PROGRAM prgVar
VAR
	fbVar			: FB_VarInfo_V3;
	fbrw1			: FB_ReadWrite_V2;
END_VAR

fbVar(
	bReadInfo:= , 
	eTMCFile:= eSelectTMCFile.eDontUseTMCFile, 
	eSavePositionTMCFile:= eSavePositionOnPLC.ePostionC, 
	udiCounterFoundVariables=> , 
	bError=> , 
	bBusy=> , 
	byProgress=> , 
	udiErrorCodeOut=> , 
	eErrorVarInfo_Out=> , 
	sVarWithError=> );
fbVar();
fbVar();	

fbRW1(	eUploadType := eSelectDataUploadType.e_Change_Intervall5min,
		bBusy=> , 
		bError=> , 
		udiErrorCodeOut=> , 
		eErrorReadWrite_Out=> );

END_PROGRAM

(* stored: Version 1.1.0.1, ProductVersion 3.1.4024.12
   POU prgVar: Id {2131ffba-df93-4f0e-b2c8-6272bbbd19d5}, SpecialFunc None *)
